// TIA Portal project "Project1" (V15.1)

(* hardware
DEVICE "S7-1200 station_1"  S7-1200 Station
   slot 0: "Rack_0"  S7-1200 Rack  Rack  V1.0
   slot 1: "PLC_1"  CPU 1215C DC/DC/DC  6ES7 215-1AG40-0XB0  V4.3
*)

// ===== PLC "PLC_1"  CPU 1215C DC/DC/DC =====

VAR_GLOBAL   // PLC tag table "Default tag table"
   "%I0.0" AT %I0.0 : Bool;
   "%I0.1" AT %I0.1 : Bool;
   "SNIMASPOSLED" AT %I0.2 : Bool;
   "KNOPKA3" AT %I0.3 : Bool;
   "%I0.4" AT %I0.4 : Bool;
   "%I0.5" AT %I0.5 : Bool;
   "KS2" AT %I0.6 : Bool;
   "SNIMAC1" AT %I0.7 : Bool;
   "KS1" AT %I1.0 : Bool;
   "%I0.9" AT %I1.1 : Bool;
   "%I0.10" AT %I1.2 : Bool;
   "%I0.11" AT %I1.3 : Bool;
   "%I0.12" AT %I1.4 : Bool;
   "%I0.13" AT %I1.5 : Bool;
   "%I0.14" AT %I1.6 : Bool;
   "%I0.15" AT %I1.7 : Bool;
   "%I0.16" AT %I2.0 : Bool;
   "%I0.17" AT %I2.1 : Bool;
   "%I0.18" AT %I2.2 : Bool;
   "%I0.19" AT %I2.3 : Bool;
   "%I0.20" AT %I2.4 : Bool;
   "%I0.21" AT %I2.5 : Bool;
   "%I0.22" AT %I2.6 : Bool;
   "%I0.23" AT %I2.7 : Bool;
   "%I0.24" AT %I3.0 : Bool;
   "%I0.25" AT %I3.1 : Bool;
   "%I0.26" AT %I3.2 : Bool;
   "%I0.27" AT %I3.3 : Bool;
   "%I0.28" AT %I3.4 : Bool;
   "%I0.29" AT %I3.5 : Bool;
   "%I0.30" AT %I3.6 : Bool;
   "%I0.31" AT %I3.7 : Bool;
   "%I0.32" AT %I4.0 : Bool;
   "%I0.33" AT %I4.1 : Bool;
   "%I0.34" AT %I4.2 : Bool;
   "%I0.35" AT %I4.3 : Bool;
   "%I0.36" AT %I4.4 : Bool;
   "%I0.37" AT %I4.5 : Bool;
   "%I0.38" AT %I4.6 : Bool;
   "%I0.39" AT %I4.7 : Bool;
   "%I0.40" AT %I5.0 : Bool;
   "%Q0.0" AT %I5.1 : Bool;
   "%Q0.1" AT %I5.2 : Bool;
   "pravypas(q02)" AT %Q0.2 : Bool;
   "%Q0.3" AT %I5.4 : Bool;
   "otocnik(q04)" AT %Q0.4 : Bool;
   "porshen3poz3" AT %Q0.5 : Bool;
   "porshen3poz5" AT %Q0.6 : Bool;
   "%Q0.7" AT %I6.0 : Bool;
   "Tag_1" AT %Q0.0 : Bool;
   "porshen1" AT %Q1.0 : Bool;
   "porshen2" AT %Q0.7 : Bool;
   "generator" AT %Q1.1 : Bool;
   "pomockapreos" AT %M0.1 : Bool;
   "pomocka2" AT %M0.2 : Bool;
   "Tag_2" AT %M99.5 : Bool;
   "Tag_3" AT %M100.1 : Bool;
   "Tag_4" AT %M100.2 : Bool;
   "STOL_OK" AT %M100.3 : Bool;
   "Tag_5" AT %M100.7 : Bool;
   "poz1_id" AT %MW20 : Int;
   "poz2_id" AT %MW22 : Int;
   "poz3_id" AT %MW24 : Int;
   "poz4_id" AT %MW26 : Int;
   "poz5_id" AT %MW28 : Int;
   "poz6_id" AT %MW30 : Int;
   "P1_pracuje" AT %M0.0 : Bool;
   "P2_pracuje" AT %M0.3 : Bool;
   "poz1" AT %M0.4 : Bool;
   "ID_objektu" AT %MW50 : Int;
   "P3_pracuje" AT %M52.0 : Bool;
   "Tag_7" AT %M60.1 : Bool;
   "P2_dopracoval" AT %M70.0 : Bool;
   "nechavanie_id" AT %MW80 : Int;
   "Tag_8" AT %M100.5 : Bool;
   "poz2" AT %M0.5 : Bool;
   "Tag_9" AT %M100.4 : Bool;
   "poz4" AT %M0.6 : Bool;
   "pomocka_pres_os" AT %M0.7 : Bool;
   "poz5" AT %M1.0 : Bool;
   "pomocka_poz3" AT %M1.1 : Bool;
   "P3_DOPRACOVAL" AT %M1.2 : Bool;
   "pozobsaden" AT %M1.3 : Bool;
   "poz3" AT %M100.6 : Bool;
   "PT" AT %M101.0 : Bool;
END_VAR

DATA_BLOCK "DATA"   // DB2
{ S7_Optimized_Access := 'TRUE' }
VERSION : 0.1
BEGIN
END_DATA_BLOCK

// folder: System blocks/Program resources

DATA_BLOCK "casovac1"   // DB1
{ S7_Optimized_Access := 'TRUE' }
AUTHOR : Simatic
FAMILY : IEC
NAME : IEC_TMR
VERSION : 1.0
// stored: InstanceOfName IEC_TIMER
"IEC_TIMER"
BEGIN
END_DATA_BLOCK

DATA_BLOCK "IEC_Timer_0_DB"   // DB3
{ S7_Optimized_Access := 'TRUE' }
AUTHOR : Simatic
FAMILY : IEC
NAME : IEC_TMR
VERSION : 1.0
// stored: InstanceOfName IEC_TIMER
"IEC_TIMER"
BEGIN
END_DATA_BLOCK

DATA_BLOCK "counter_pre_porshen2"   // DB4
{ S7_Optimized_Access := 'TRUE' }
AUTHOR : Simatic
FAMILY : IEC
NAME : CNTR
VERSION : 1.0
// stored: InstanceOfName IEC_COUNTER
"IEC_COUNTER"
BEGIN
END_DATA_BLOCK

DATA_BLOCK "IEC_Timer_0_DB_1"   // DB5
{ S7_Optimized_Access := 'TRUE' }
AUTHOR : Simatic
FAMILY : IEC
NAME : IEC_TMR
VERSION : 1.0
// stored: InstanceOfName IEC_TIMER
"IEC_TIMER"
BEGIN
END_DATA_BLOCK

DATA_BLOCK "casovac3"   // DB6
{ S7_Optimized_Access := 'TRUE' }
AUTHOR : Simatic
FAMILY : IEC
NAME : IEC_TMR
VERSION : 1.0
// stored: InstanceOfName IEC_TIMER
"IEC_TIMER"
BEGIN
END_DATA_BLOCK

DATA_BLOCK "casovacpoz3"   // DB8
{ S7_Optimized_Access := 'TRUE' }
AUTHOR : Simatic
FAMILY : IEC
NAME : IEC_TMR
VERSION : 1.0
// stored: InstanceOfName IEC_TIMER
"IEC_TIMER"
BEGIN
END_DATA_BLOCK

DATA_BLOCK "IEC_Timer_0_DB_2"   // DB10
{ S7_Optimized_Access := 'TRUE' }
AUTHOR : Simatic
FAMILY : IEC
NAME : IEC_TMR
VERSION : 1.0
// stored: InstanceOfName IEC_TIMER
"IEC_TIMER"
BEGIN
END_DATA_BLOCK

DATA_BLOCK "casovac5"   // DB12
{ S7_Optimized_Access := 'TRUE' }
AUTHOR : Simatic
FAMILY : IEC
NAME : IEC_TMR
VERSION : 1.0
// stored: InstanceOfName IEC_TIMER
"IEC_TIMER"
BEGIN
END_DATA_BLOCK

// folder: (top level)

ORGANIZATION_BLOCK "Main"   // OB1, LAD, ProgramCycle
TITLE = "Main Program Sweep (Cycle)"
{ S7_Optimized_Access := 'TRUE' }
VERSION : 0.1
   VAR_INPUT
      Initial_Call : Bool;   // Initial call of this OB
      Remanence : Bool;   // =True, if remanent data are available
   END_VAR
   VAR_TEMP   // added for the SCL form of the ladder/FBD networks
      _w1 : Bool;
      _w2 : Bool;
   END_VAR
BEGIN

REGION Network 1: main
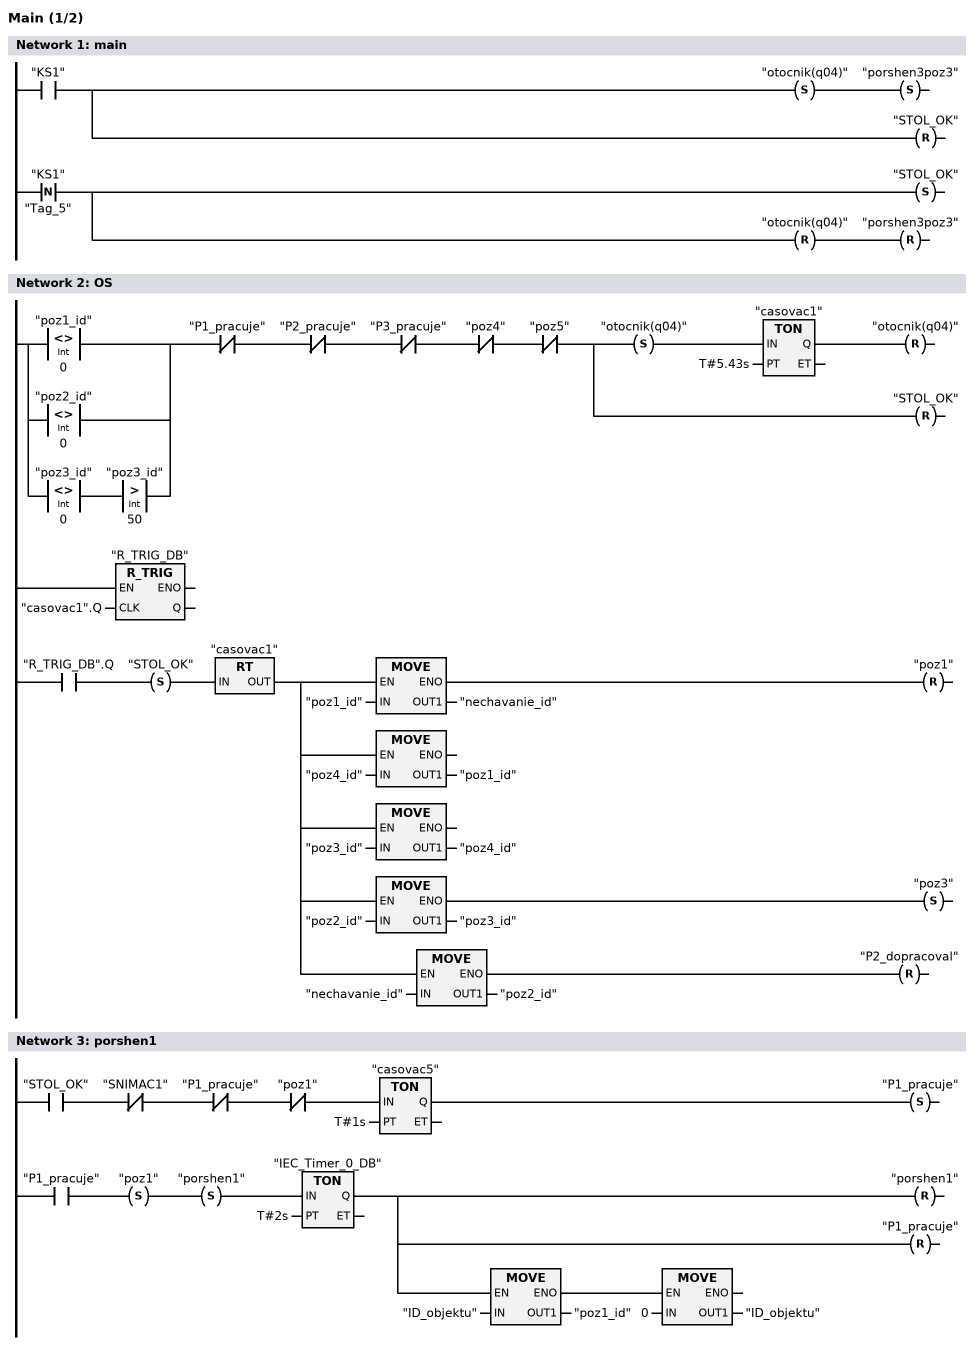
   RUNG wire#powerrail
      Contact( "KS1" )
      wire#w1
      S_Coil( "otocnik(q04)" )
      S_Coil( "porshen3poz3" )
   END_RUNG
   RUNG wire#w1
      R_Coil( "STOL_OK" )
   END_RUNG
   RUNG wire#powerrail
      N_Contact(operand := "KS1", bit := "Tag_5")
      wire#w2
      S_Coil( "STOL_OK" )
   END_RUNG
   RUNG wire#w2
      R_Coil( "otocnik(q04)" )
      R_Coil( "porshen3poz3" )
   END_RUNG
   // the same network as SCL:
   IF "KS1" THEN
       "otocnik(q04)" := TRUE;
       "porshen3poz3" := TRUE;
       "STOL_OK" := FALSE;
   END_IF;
   #_w1 := NOT "KS1" AND "Tag_5";   // falling edge of "KS1"
   "Tag_5" := "KS1";
   IF #_w1 THEN
       "STOL_OK" := TRUE;
       "otocnik(q04)" := FALSE;
       "porshen3poz3" := FALSE;
   END_IF;
END_REGION

REGION Network 2: OS
   #_w1 := (("poz1_id" <> 0) OR ("poz2_id" <> 0) OR (("poz3_id" <> 0) AND ("poz3_id" > 50))) AND NOT "P1_pracuje" AND NOT "P2_pracuje" AND NOT "P3_pracuje" AND NOT "poz4" AND NOT "poz5";
   IF #_w1 THEN "otocnik(q04)" := TRUE; END_IF;
   "casovac1".TON(IN := #_w1, PT := T#5.43s);
   IF "casovac1".Q THEN "otocnik(q04)" := FALSE; END_IF;
   IF #_w1 THEN "STOL_OK" := FALSE; END_IF;
   "R_TRIG_DB"(CLK := "casovac1".Q);   // R_TRIG
   IF "R_TRIG_DB".Q THEN
       "STOL_OK" := TRUE;
       RESET_TIMER("casovac1");
       "nechavanie_id" := "poz1_id";
       "poz1" := FALSE;
       "poz1_id" := "poz4_id";
       "poz4_id" := "poz3_id";
       "poz3_id" := "poz2_id";
       "poz3" := TRUE;
       "poz2_id" := "nechavanie_id";
       "P2_dopracoval" := FALSE;
   END_IF;
END_REGION

REGION Network 3: porshen1
   "casovac5".TON(IN := "STOL_OK" AND NOT "SNIMAC1" AND NOT "P1_pracuje" AND NOT "poz1", PT := T#1s);
   IF "casovac5".Q THEN "P1_pracuje" := TRUE; END_IF;
   IF "P1_pracuje" THEN
       "poz1" := TRUE;
       "porshen1" := TRUE;
   END_IF;
   "IEC_Timer_0_DB".TON(IN := "P1_pracuje", PT := T#2s);
   IF "IEC_Timer_0_DB".Q THEN
       "porshen1" := FALSE;
       "P1_pracuje" := FALSE;
       "poz1_id" := "ID_objektu";
       "ID_objektu" := 0;
   END_IF;
END_REGION

REGION Network 4: porshen2
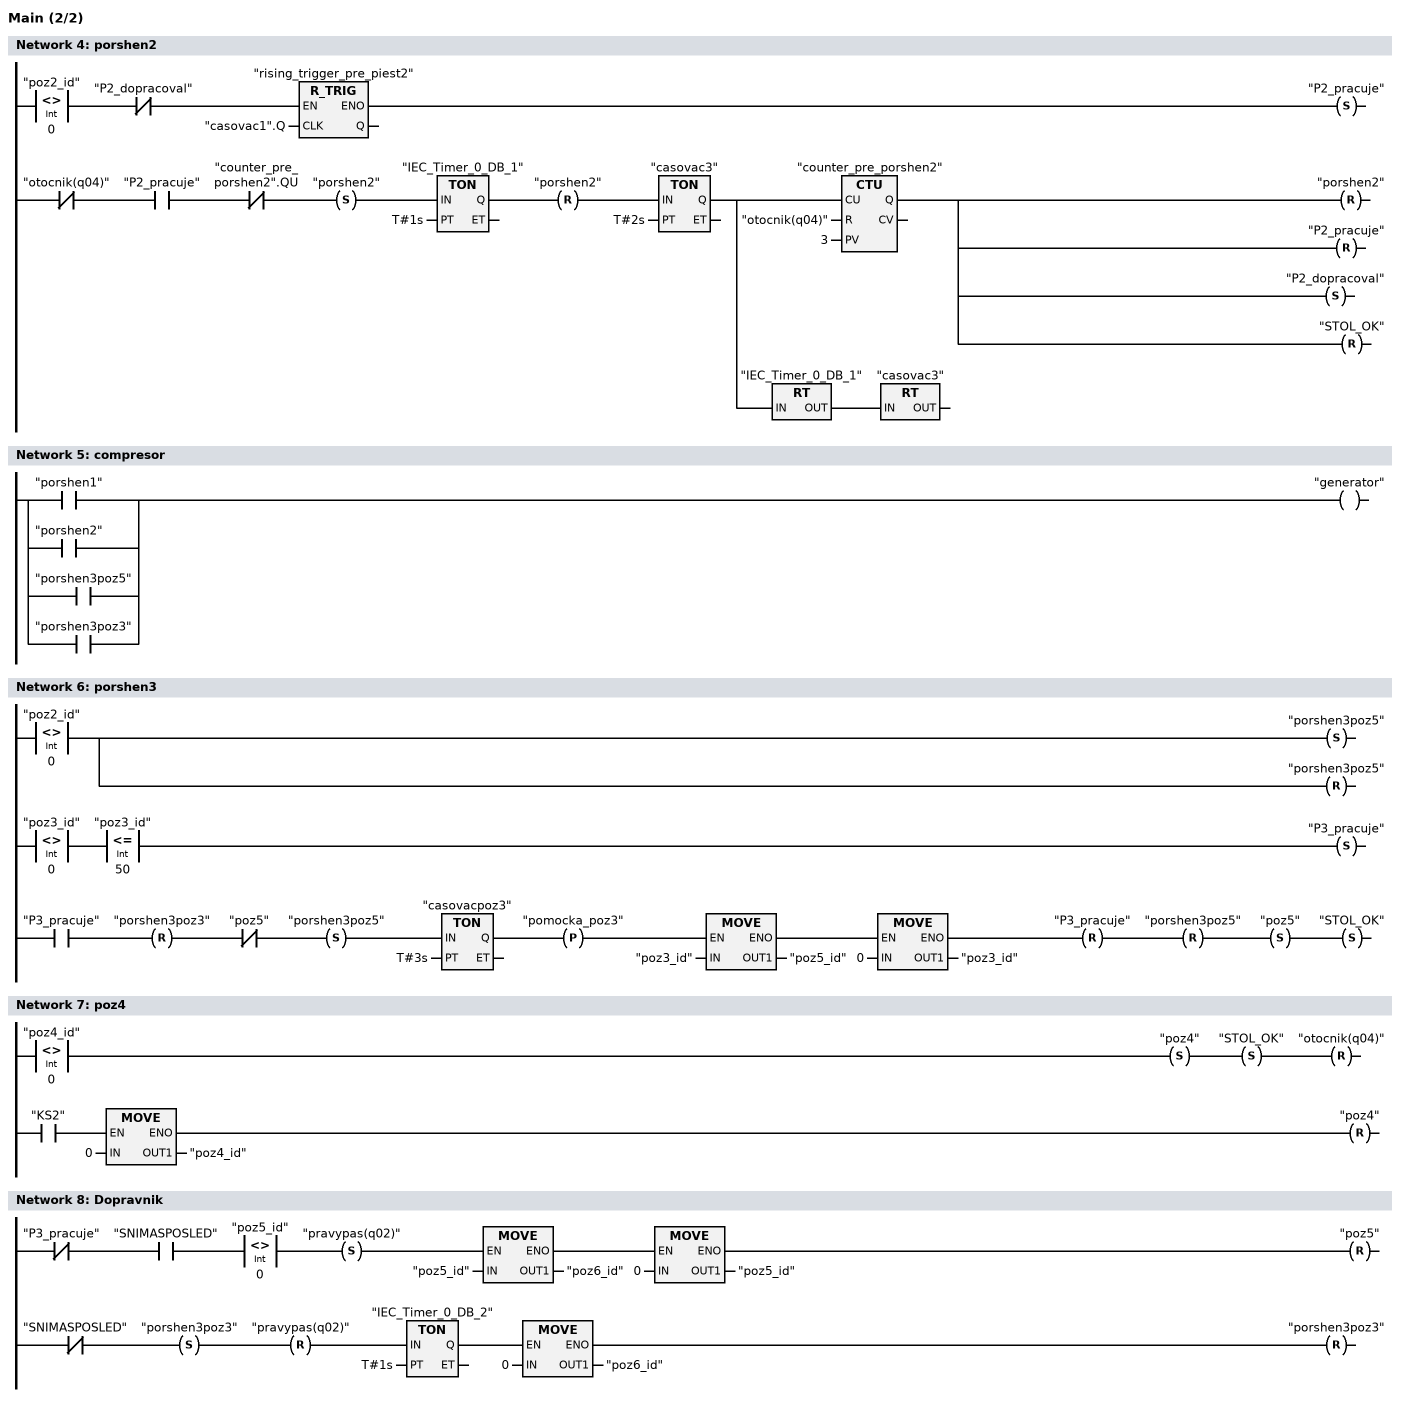
   // ENO of a box is taken as its EN; it also drops when the box reports an error
   IF ("poz2_id" <> 0) AND NOT "P2_dopracoval" THEN
       "rising_trigger_pre_piest2"(CLK := "casovac1".Q);   // R_TRIG
       "P2_pracuje" := TRUE;
   END_IF;
   #_w1 := NOT "otocnik(q04)" AND "P2_pracuje" AND NOT "counter_pre_porshen2".QU;
   IF #_w1 THEN "porshen2" := TRUE; END_IF;
   "IEC_Timer_0_DB_1".TON(IN := #_w1, PT := T#1s);
   IF "IEC_Timer_0_DB_1".Q THEN "porshen2" := FALSE; END_IF;
   "casovac3".TON(IN := "IEC_Timer_0_DB_1".Q, PT := T#2s);
   "counter_pre_porshen2".CTU(CU := "casovac3".Q, R := "otocnik(q04)", PV := 3);
   IF "counter_pre_porshen2".Q THEN
       "porshen2" := FALSE;
       "P2_pracuje" := FALSE;
       "P2_dopracoval" := TRUE;
       "STOL_OK" := FALSE;
   END_IF;
   IF "casovac3".Q THEN
       RESET_TIMER("IEC_Timer_0_DB_1");
       RESET_TIMER("casovac3");
   END_IF;
END_REGION

REGION Network 5: compresor
   RUNG wire#powerrail
      Contact( "porshen1" )
      wire#w1
      Coil( "generator" )
   END_RUNG
   RUNG wire#powerrail
      Contact( "porshen2" )
   END_RUNG wire#w1
   RUNG wire#powerrail
      Contact( "porshen3poz5" )
   END_RUNG wire#w1
   RUNG wire#powerrail
      Contact( "porshen3poz3" )
   END_RUNG wire#w1
   // the same network as SCL:
   "generator" := "porshen1" OR "porshen2" OR "porshen3poz5" OR "porshen3poz3";
END_REGION

REGION Network 6: porshen3
   IF "poz2_id" <> 0 THEN
       "porshen3poz5" := TRUE;
       "porshen3poz5" := FALSE;
   END_IF;
   IF ("poz3_id" <> 0) AND ("poz3_id" <= 50) THEN "P3_pracuje" := TRUE; END_IF;
   IF "P3_pracuje" THEN "porshen3poz3" := FALSE; END_IF;
   #_w1 := "P3_pracuje" AND NOT "poz5";
   IF #_w1 THEN "porshen3poz5" := TRUE; END_IF;
   "casovacpoz3".TON(IN := #_w1, PT := T#3s);
   #_w2 := "casovacpoz3".Q AND NOT "pomocka_poz3";   // rising edge
   "pomocka_poz3" := "casovacpoz3".Q;
   IF #_w2 THEN
       "poz5_id" := "poz3_id";
       "poz3_id" := 0;
       "P3_pracuje" := FALSE;
       "porshen3poz5" := FALSE;
       "poz5" := TRUE;
       "STOL_OK" := TRUE;
   END_IF;
END_REGION

REGION Network 7: poz4
   RUNG wire#powerrail
      { S7_Templates := "SrcType := Int" } NE_Contact(in1 := "poz4_id", in2 := 0)
      S_Coil( "poz4" )
      S_Coil( "STOL_OK" )
      R_Coil( "otocnik(q04)" )
   END_RUNG
   RUNG wire#powerrail
      Contact( "KS2" )
      Move(in := 0, out1 => "poz4_id")
      R_Coil( "poz4" )
   END_RUNG
   // the same network as SCL:
   IF "poz4_id" <> 0 THEN
       "poz4" := TRUE;
       "STOL_OK" := TRUE;
       "otocnik(q04)" := FALSE;
   END_IF;
   IF "KS2" THEN
       "poz4_id" := 0;
       "poz4" := FALSE;
   END_IF;
END_REGION

REGION Network 8: Dopravnik
   IF NOT "P3_pracuje" AND "SNIMASPOSLED" AND ("poz5_id" <> 0) THEN
       "pravypas(q02)" := TRUE;
       "poz6_id" := "poz5_id";
   END_IF;
   #_w1 := NOT "P3_pracuje" AND "SNIMASPOSLED" AND ("poz5_id" <> 0);
   IF #_w1 THEN
       "poz5_id" := 0;
       "poz5" := FALSE;
   END_IF;
   IF NOT "SNIMASPOSLED" THEN
       "porshen3poz3" := TRUE;
       "pravypas(q02)" := FALSE;
   END_IF;
   "IEC_Timer_0_DB_2".TON(IN := NOT "SNIMASPOSLED", PT := T#1s);
   IF "IEC_Timer_0_DB_2".Q THEN
       "poz6_id" := 0;
       "porshen3poz3" := FALSE;
   END_IF;
END_REGION

REGION Network 9: poz3
END_REGION
END_ORGANIZATION_BLOCK